FUNCTION_BLOCK FbSealedinCoil
VAR_INPUT
	xTrigger: BOOL;
END_VAR
VAR_OUTPUT
	xSealedInCoil: BOOL;
END_VAR

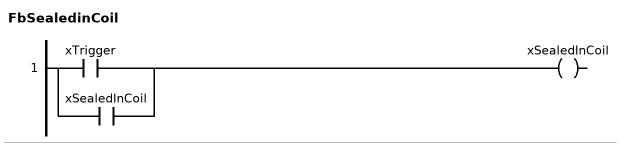
// NETWORK 1
xSealedInCoil := xTrigger OR xSealedInCoil;

END_FUNCTION_BLOCK

(* stored: Version 1.1.0.1, ProductVersion 3.1.4024.12
   POU FbSealedinCoil: Id {7a4669b7-f0b3-498b-8cc7-ebcb19d806ca}, SpecialFunc None *)
